TYPE ST_TopElement1_HMI_Link EXTENDS ST_BaseTopElement_HMI_Link :
STRUCT
	stTopElement		: ST_TopElement1_HMI;
	
	
END_STRUCT
END_TYPE

(* stored: Version 1.1.0.1, ProductVersion 3.1.4024.15
   DUT ST_TopElement1_HMI_Link: Id {afb6776f-e6d0-4d3c-85b9-064d0107abb6} *)
